% RSLogix 500 project Sesion10_Tarea1_Josue Santana Robledo Corona.RSS, saved by version 8.40.00.08 %
PROJECT "UNTITLED"    % processor: MicroLogix 1200 %

PROGRAM FILES
  LAD 2 "MAIN"  6 rungs
  LAD 3 "ENTRADAS"  9 rungs
  LAD 4 "SALIDAS"  6 rungs
  LAD 5 "ALARMAS"  1 rungs
  LAD 6 "MANUAL"  6 rungs
  LAD 7 "AUTOMATICO"  16 rungs
  LAD 8 "HMI"  1 rungs
  LAD 9 "LS"  3 rungs

DATA FILES
  O0 OUTPUT  4 elements
  I1 INPUT  4 elements
  S2 STATUS  66 elements
  B3 BINARY  3 elements
  T4 TIMER  3 elements
  C5 COUNTER  1 elements
  R6 CONTROL  1 elements
  N7 INTEGER  1 elements
  F8 FLOAT  1 elements

LADDER 2 "MAIN"
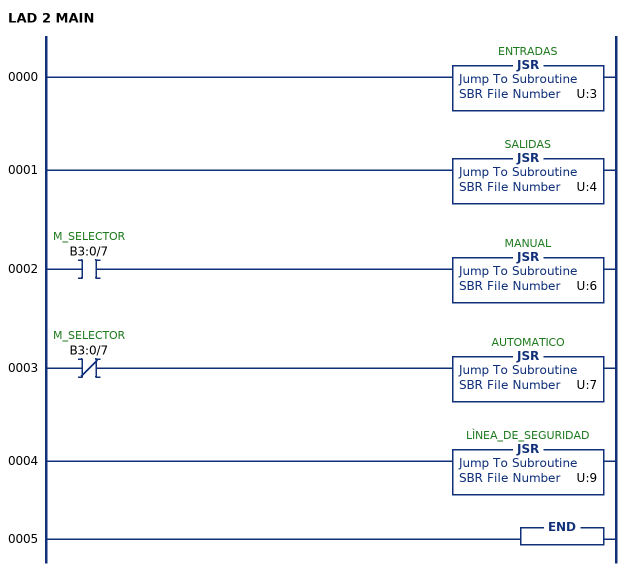
% Rung: 0 %
SOR JSR U:3 EOR
%   U:3  ENTRADAS %
% Rung: 1 %
SOR JSR U:4 EOR
%   U:4  SALIDAS %
% Rung: 2 %
SOR XIC B3:0/7 JSR U:6 EOR
%   B3:0/7  M_SELECTOR %
%   U:6  MANUAL %
% Rung: 3 %
SOR XIO B3:0/7 JSR U:7 EOR
%   B3:0/7  M_SELECTOR %
%   U:7  AUTOMATICO %
% Rung: 4 %
SOR JSR U:9 EOR
%   U:9  LÌNEA_DE_SEGURIDAD %
% Rung: 5 %
SOR END EOR

LADDER 3 "ENTRADAS"
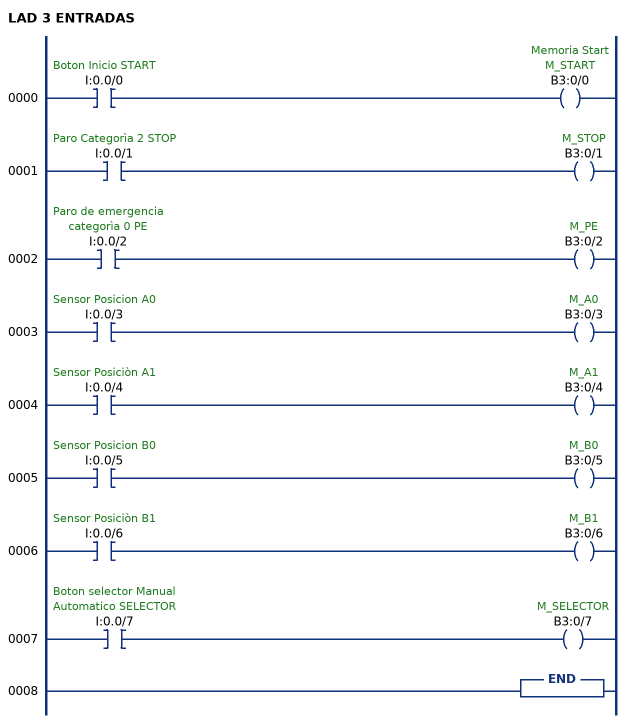
% Rung: 0 %
SOR XIC I:0.0/0 OTE B3:0/0 EOR
%   I:0.0/0  START  "Boton Inicio" %
%   B3:0/0  M_START  "Memoria Start" %
% Rung: 1 %
SOR XIC I:0.0/1 OTE B3:0/1 EOR
%   I:0.0/1  STOP  "Paro Categorìa 2" %
%   B3:0/1  M_STOP %
% Rung: 2 %
SOR XIC I:0.0/2 OTE B3:0/2 EOR
%   I:0.0/2  PE  "Paro de emergencia categorìa 0" %
%   B3:0/2  M_PE %
% Rung: 3 %
SOR XIC I:0.0/3 OTE B3:0/3 EOR
%   I:0.0/3  A0  "Sensor Posicion" %
%   B3:0/3  M_A0 %
% Rung: 4 %
SOR XIC I:0.0/4 OTE B3:0/4 EOR
%   I:0.0/4  A1  "Sensor Posiciòn" %
%   B3:0/4  M_A1 %
% Rung: 5 %
SOR XIC I:0.0/5 OTE B3:0/5 EOR
%   I:0.0/5  B0  "Sensor Posicion" %
%   B3:0/5  M_B0 %
% Rung: 6 %
SOR XIC I:0.0/6 OTE B3:0/6 EOR
%   I:0.0/6  B1  "Sensor Posiciòn" %
%   B3:0/6  M_B1 %
% Rung: 7 %
SOR XIC I:0.0/7 OTE B3:0/7 EOR
%   I:0.0/7  SELECTOR  "Boton selector Manual Automatico" %
%   B3:0/7  M_SELECTOR %
% Rung: 8 %
SOR END EOR

LADDER 4 "SALIDAS"
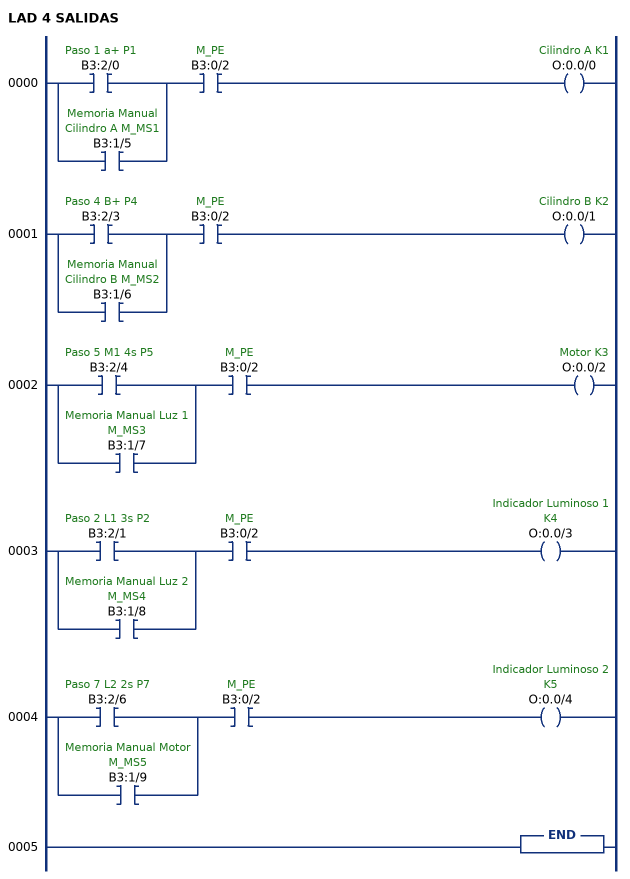
% Rung: 0 %
SOR BST XIC B3:2/0 NXB XIC B3:1/5 BND XIC B3:0/2 OTE O:0.0/0 EOR
%   B3:2/0  P1  "Paso 1 a+" %
%   B3:1/5  M_MS1  "Memoria Manual Cilindro A" %
%   B3:0/2  M_PE %
%   O:0.0/0  K1  "Cilindro A" %
% Rung: 1 %
SOR BST XIC B3:2/3 NXB XIC B3:1/6 BND XIC B3:0/2 OTE O:0.0/1 EOR
%   B3:2/3  P4  "Paso 4 B+" %
%   B3:1/6  M_MS2  "Memoria Manual Cilindro B" %
%   B3:0/2  M_PE %
%   O:0.0/1  K2  "Cilindro B" %
% Rung: 2 %  % edit flag set %
SOR BST XIC B3:2/4 NXB XIC B3:1/7 BND XIC B3:0/2 OTE O:0.0/2 EOR
%   B3:2/4  P5  "Paso 5 M1 4s" %
%   B3:1/7  M_MS3  "Memoria Manual Luz 1" %
%   B3:0/2  M_PE %
%   O:0.0/2  K3  "Motor" %
% Rung: 3 %  % edit flag set %
SOR BST XIC B3:2/1 NXB XIC B3:1/8 BND XIC B3:0/2 OTE O:0.0/3 EOR
%   B3:2/1  P2  "Paso 2 L1 3s" %
%   B3:1/8  M_MS4  "Memoria Manual Luz 2" %
%   B3:0/2  M_PE %
%   O:0.0/3  K4  "Indicador Luminoso 1" %
% Rung: 4 %  % edit flag set %
SOR BST XIC B3:2/6 NXB XIC B3:1/9 BND XIC B3:0/2 OTE O:0.0/4 EOR
%   B3:2/6  P7  "Paso 7 L2 2s" %
%   B3:1/9  M_MS5  "Memoria Manual Motor" %
%   B3:0/2  M_PE %
%   O:0.0/4  K5  "Indicador Luminoso 2" %
% Rung: 5 %
SOR END EOR

LADDER 6 "MANUAL"
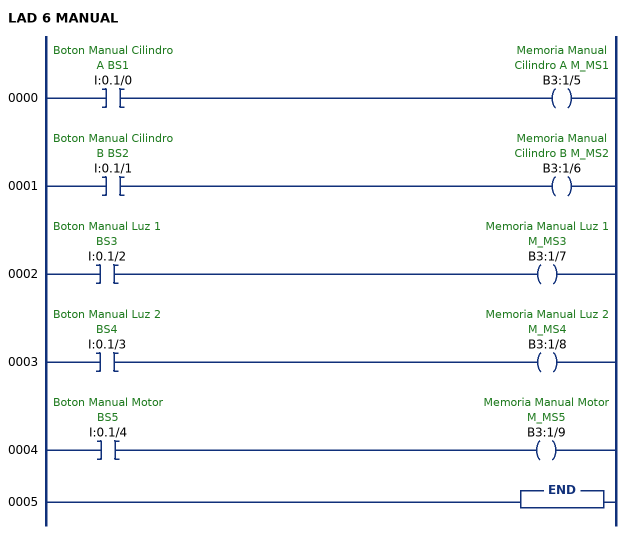
% Rung: 0 %
SOR XIC I:0.1/0 OTE B3:1/5 EOR
%   I:0.1/0  BS1  "Boton Manual Cilindro A" %
%   B3:1/5  M_MS1  "Memoria Manual Cilindro A" %
% Rung: 1 %
SOR XIC I:0.1/1 OTE B3:1/6 EOR
%   I:0.1/1  BS2  "Boton Manual Cilindro B" %
%   B3:1/6  M_MS2  "Memoria Manual Cilindro B" %
% Rung: 2 %
SOR XIC I:0.1/2 OTE B3:1/7 EOR
%   I:0.1/2  BS3  "Boton Manual Luz 1" %
%   B3:1/7  M_MS3  "Memoria Manual Luz 1" %
% Rung: 3 %
SOR XIC I:0.1/3 OTE B3:1/8 EOR
%   I:0.1/3  BS4  "Boton Manual Luz 2" %
%   B3:1/8  M_MS4  "Memoria Manual Luz 2" %
% Rung: 4 %
SOR XIC I:0.1/4 OTE B3:1/9 EOR
%   I:0.1/4  BS5  "Boton Manual Motor" %
%   B3:1/9  M_MS5  "Memoria Manual Motor" %
% Rung: 5 %
SOR END EOR

LADDER 7 "AUTOMATICO"
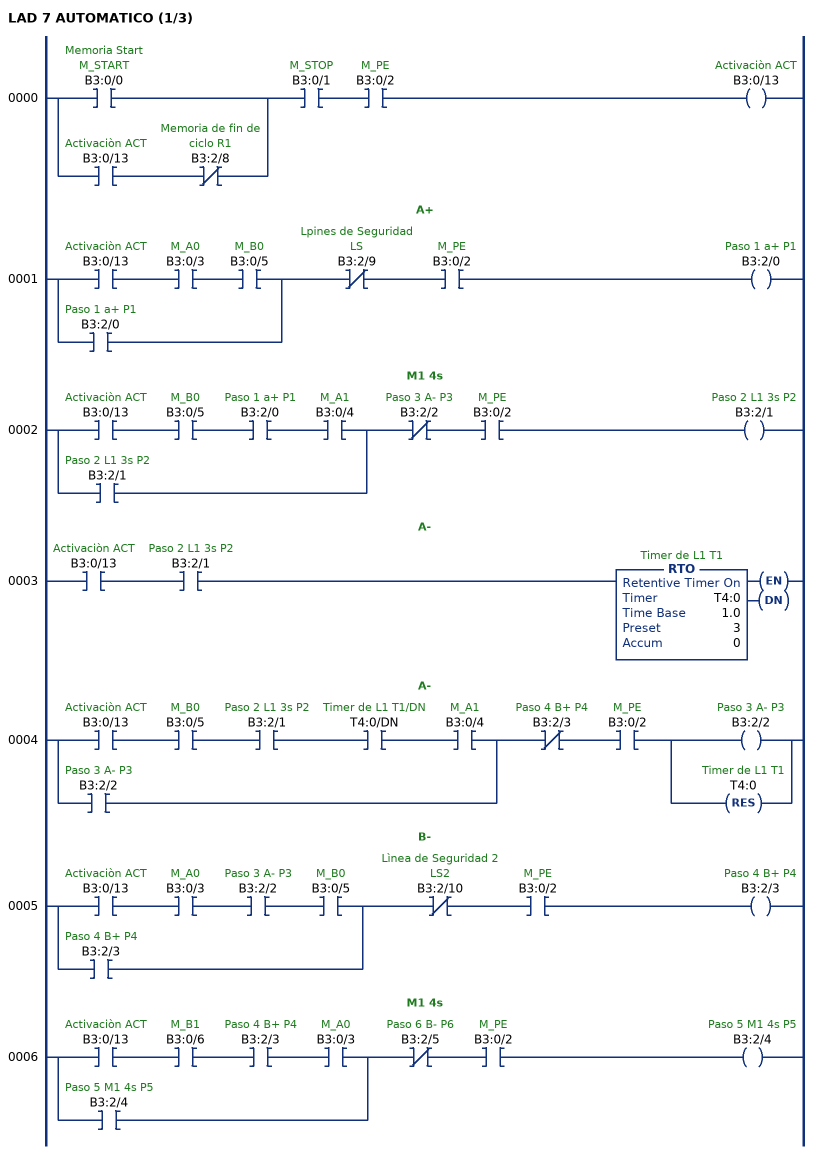
% Rung: 0 %
SOR BST XIC B3:0/0 NXB XIC B3:0/13 XIO B3:2/8 BND XIC B3:0/1 XIC B3:0/2 OTE B3:0/13 EOR
%   B3:0/0  M_START  "Memoria Start" %
%   B3:0/13  ACT  "Activaciòn" %
%   B3:2/8  R1  "Memoria de fin de ciclo" %
%   B3:0/1  M_STOP %
%   B3:0/2  M_PE %
% Rung: 1 %  % edit flag set %
% TITLE: A+ %
SOR BST XIC B3:0/13 XIC B3:0/3 XIC B3:0/5 NXB XIC B3:2/0 BND XIO B3:2/9 XIC B3:0/2 OTE B3:2/0 EOR
%   B3:0/13  ACT  "Activaciòn" %
%   B3:0/3  M_A0 %
%   B3:0/5  M_B0 %
%   B3:2/0  P1  "Paso 1 a+" %
%   B3:2/9  LS  "Lpines de Seguridad" %
%   B3:0/2  M_PE %
% Rung: 2 %
% TITLE: M1 4s %
SOR BST XIC B3:0/13 XIC B3:0/5 XIC B3:2/0 XIC B3:0/4 NXB XIC B3:2/1 BND XIO B3:2/2 XIC B3:0/2 OTE B3:2/1 EOR
%   B3:0/13  ACT  "Activaciòn" %
%   B3:0/5  M_B0 %
%   B3:2/0  P1  "Paso 1 a+" %
%   B3:0/4  M_A1 %
%   B3:2/1  P2  "Paso 2 L1 3s" %
%   B3:2/2  P3  "Paso 3 A-" %
%   B3:0/2  M_PE %
% Rung: 3 %
% TITLE: A- %
SOR XIC B3:0/13 XIC B3:2/1 RTO T4:0 1.0 3 0 EOR
%   B3:0/13  ACT  "Activaciòn" %
%   B3:2/1  P2  "Paso 2 L1 3s" %
%   T4:0  T1  "Timer de L1" %
% Rung: 4 %
% TITLE: A- %
SOR BST XIC B3:0/13 XIC B3:0/5 XIC B3:2/1 XIC T4:0/DN XIC B3:0/4 NXB XIC B3:2/2 BND XIO B3:2/3 XIC B3:0/2 BST OTE B3:2/2 NXB RES T4:0 BND EOR
%   B3:0/13  ACT  "Activaciòn" %
%   B3:0/5  M_B0 %
%   B3:2/1  P2  "Paso 2 L1 3s" %
%   T4:0  T1  "Timer de L1" %
%   B3:0/4  M_A1 %
%   B3:2/2  P3  "Paso 3 A-" %
%   B3:2/3  P4  "Paso 4 B+" %
%   B3:0/2  M_PE %
% Rung: 5 %  % edit flag set %
% TITLE: B- %
SOR BST XIC B3:0/13 XIC B3:0/3 XIC B3:2/2 XIC B3:0/5 NXB XIC B3:2/3 BND XIO B3:2/10 XIC B3:0/2 OTE B3:2/3 EOR
%   B3:0/13  ACT  "Activaciòn" %
%   B3:0/3  M_A0 %
%   B3:2/2  P3  "Paso 3 A-" %
%   B3:0/5  M_B0 %
%   B3:2/3  P4  "Paso 4 B+" %
%   B3:2/10  LS2  "Lìnea de Seguridad 2" %
%   B3:0/2  M_PE %
% Rung: 6 %
% TITLE: M1 4s %
SOR BST XIC B3:0/13 XIC B3:0/6 XIC B3:2/3 XIC B3:0/3 NXB XIC B3:2/4 BND XIO B3:2/5 XIC B3:0/2 OTE B3:2/4 EOR
%   B3:0/13  ACT  "Activaciòn" %
%   B3:0/6  M_B1 %
%   B3:2/3  P4  "Paso 4 B+" %
%   B3:0/3  M_A0 %
%   B3:2/4  P5  "Paso 5 M1 4s" %
%   B3:2/5  P6  "Paso 6 B-" %
%   B3:0/2  M_PE %

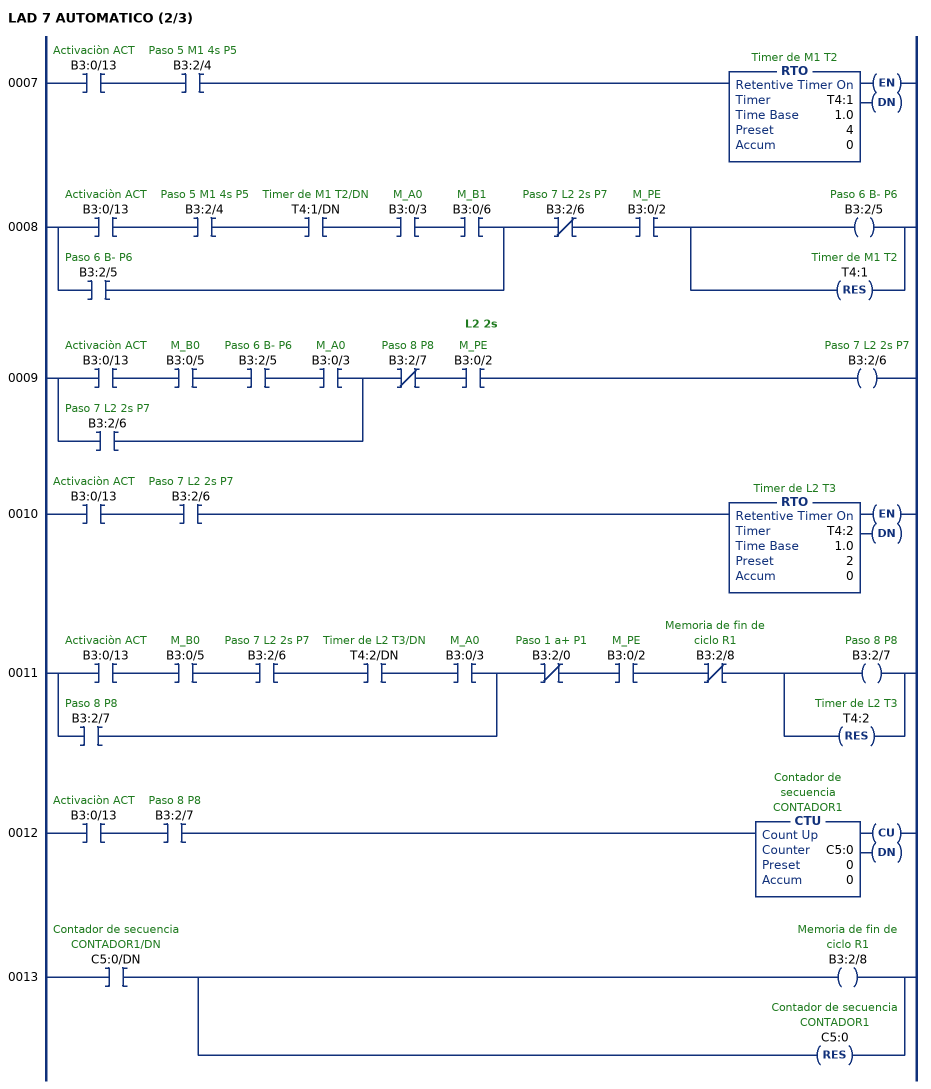
% Rung: 7 %
SOR XIC B3:0/13 XIC B3:2/4 RTO T4:1 1.0 4 0 EOR
%   B3:0/13  ACT  "Activaciòn" %
%   B3:2/4  P5  "Paso 5 M1 4s" %
%   T4:1  T2  "Timer de M1" %
% Rung: 8 %
SOR BST XIC B3:0/13 XIC B3:2/4 XIC T4:1/DN XIC B3:0/3 XIC B3:0/6 NXB XIC B3:2/5 BND XIO B3:2/6 XIC B3:0/2 BST OTE B3:2/5 NXB RES T4:1 BND EOR
%   B3:0/13  ACT  "Activaciòn" %
%   B3:2/4  P5  "Paso 5 M1 4s" %
%   T4:1  T2  "Timer de M1" %
%   B3:0/3  M_A0 %
%   B3:0/6  M_B1 %
%   B3:2/5  P6  "Paso 6 B-" %
%   B3:2/6  P7  "Paso 7 L2 2s" %
%   B3:0/2  M_PE %
% Rung: 9 %
% TITLE: L2 2s %
SOR BST XIC B3:0/13 XIC B3:0/5 XIC B3:2/5 XIC B3:0/3 NXB XIC B3:2/6 BND XIO B3:2/7 XIC B3:0/2 OTE B3:2/6 EOR
%   B3:0/13  ACT  "Activaciòn" %
%   B3:0/5  M_B0 %
%   B3:2/5  P6  "Paso 6 B-" %
%   B3:0/3  M_A0 %
%   B3:2/6  P7  "Paso 7 L2 2s" %
%   B3:2/7  P8  "Paso 8" %
%   B3:0/2  M_PE %
% Rung: 10 %
SOR XIC B3:0/13 XIC B3:2/6 RTO T4:2 1.0 2 0 EOR
%   B3:0/13  ACT  "Activaciòn" %
%   B3:2/6  P7  "Paso 7 L2 2s" %
%   T4:2  T3  "Timer de L2" %
% Rung: 11 %  % edit flag set %
SOR BST XIC B3:0/13 XIC B3:0/5 XIC B3:2/6 XIC T4:2/DN XIC B3:0/3 NXB XIC B3:2/7 BND XIO B3:2/0 XIC B3:0/2 XIO B3:2/8 BST OTE B3:2/7 NXB RES T4:2 BND EOR
%   B3:0/13  ACT  "Activaciòn" %
%   B3:0/5  M_B0 %
%   B3:2/6  P7  "Paso 7 L2 2s" %
%   T4:2  T3  "Timer de L2" %
%   B3:0/3  M_A0 %
%   B3:2/7  P8  "Paso 8" %
%   B3:2/0  P1  "Paso 1 a+" %
%   B3:0/2  M_PE %
%   B3:2/8  R1  "Memoria de fin de ciclo" %
% Rung: 12 %
SOR XIC B3:0/13 XIC B3:2/7 CTU C5:0 0 0 EOR
%   B3:0/13  ACT  "Activaciòn" %
%   B3:2/7  P8  "Paso 8" %
%   C5:0  CONTADOR1  "Contador de secuencia" %
% Rung: 13 %
SOR XIC C5:0/DN BST OTE B3:2/8 NXB RES C5:0 BND EOR
%   C5:0  CONTADOR1  "Contador de secuencia" %
%   B3:2/8  R1  "Memoria de fin de ciclo" %

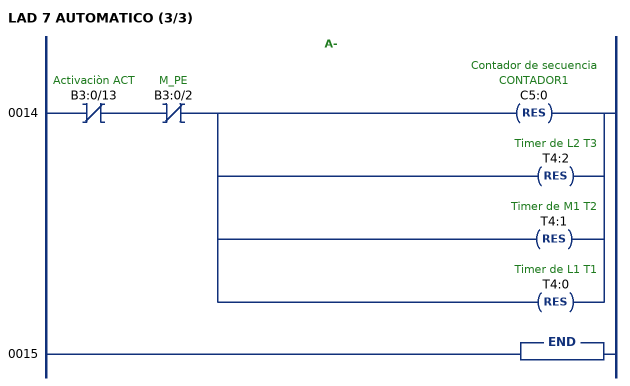
% Rung: 14 %
% TITLE: A- %
SOR XIO B3:0/13 XIO B3:0/2 BST RES C5:0 NXB BST RES T4:2 NXB BST RES T4:1 NXB RES T4:0 BND BND BND EOR
%   B3:0/13  ACT  "Activaciòn" %
%   B3:0/2  M_PE %
%   C5:0  CONTADOR1  "Contador de secuencia" %
%   T4:2  T3  "Timer de L2" %
%   T4:1  T2  "Timer de M1" %
%   T4:0  T1  "Timer de L1" %
% Rung: 15 %
SOR END EOR

LADDER 9 "LS"
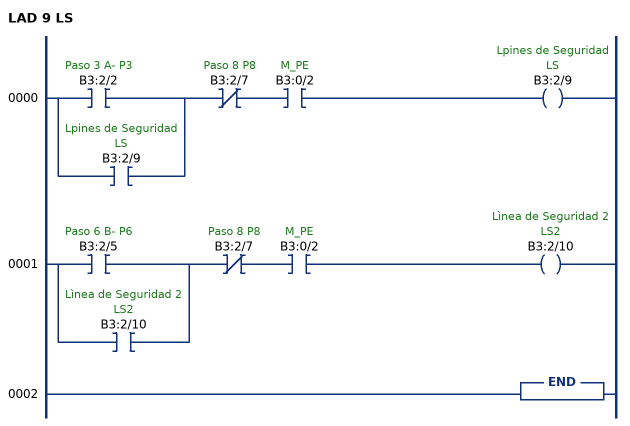
% Rung: 0 %
SOR BST XIC B3:2/2 NXB XIC B3:2/9 BND XIO B3:2/7 XIC B3:0/2 OTE B3:2/9 EOR
%   B3:2/2  P3  "Paso 3 A-" %
%   B3:2/9  LS  "Lpines de Seguridad" %
%   B3:2/7  P8  "Paso 8" %
%   B3:0/2  M_PE %
% Rung: 1 %  % edit flag set %
SOR BST XIC B3:2/5 NXB XIC B3:2/10 BND XIO B3:2/7 XIC B3:0/2 OTE B3:2/10 EOR
%   B3:2/5  P6  "Paso 6 B-" %
%   B3:2/10  LS2  "Lìnea de Seguridad 2" %
%   B3:2/7  P8  "Paso 8" %
%   B3:0/2  M_PE %
% Rung: 2 %
SOR END EOR

OTHER DOCUMENTED ADDRESSES
  B3:0/8  M_S1  "Cilindro A"
  B3:0/9  M_S2  "Cilindro B"
  B3:0/10  M_S3  "Luz 1"
  B3:0/11  M_S4  "Luz 2"
  B3:0/12  M_S5  "Motor"
  B3:1/0  M_K1  "Cilindro A"
  B3:1/1  M_K2  "Memoria Cilindro B"
  B3:1/2  M_K3  "Memoria Motor"
  B3:1/3  M_K4  "Memoria Indicador Luminoso 1"
  B3:1/4  M_K5  "Memoria Indicador Luminoso 2"

COMMENTS NOT ATTACHED TO A CURRENT RUNG
  B3:2/2: A-

DATA TABLE (non-zero values as saved)
DATA B3
% B3:0 % 0X0000 0X0000 0X0100
DATA T4
% .PRE .ACC %
% T4:0 % 3 0
% T4:1 % 4 0
% T4:2 % 2 0
